FUNCTION_BLOCK Delay2s
VAR_INPUT
	input : BOOL;
	ONdelayPT : TIME := T#2S;
END_VAR
VAR_OUTPUT
	output : BOOL;
	ONdelayET : BOOL;
END_VAR
VAR
	ONdelay : TON;
	iCount : INT;
END_VAR

ONdelay(IN:=input, PT:=ONdelayPT);

IF ONdelay.Q THEN
     iCount:= iCount+1;
     Ondelay(IN:= FALSE);

     //optional if want to keep the timer timing
     //ONdelay(IN:=input);
END_IF;

output := ONdelay.Q;

END_FUNCTION_BLOCK

(* stored: Version 1.1.0.1, ProductVersion 3.1.4024.11
   POU Delay2s: Id {655dd55a-49e9-43e5-b293-13c0abde3e61}, SpecialFunc None *)
